TYPE E_IndexPowMeas :
//Index-value connection of the second output of the power measurement terminal
(ApparantPower, ReactivePower, Energy, cosPhi, Frequency, negEnergy);
END_TYPE

(* stored: Version 1.1.0.1, ProductVersion 3.1.4018.2
   DUT E_IndexPowMeas: Id {bb2bc3b5-6309-4e15-b462-c96fa5df35ad} *)
